// TIA Portal project "Banda_Asamblare" (V15.1)

(* hardware
DEVICE "S71500/ET200MP station_1"  S7-1500 station
   slot 0: "Rail_0"  Rack  6ES7 590-1***0-0AA0
   slot 1: "PLC_1"  CPU 1513-1 PN  6ES7 513-1AL02-0AB0  V2.6
      slot 3: "CPU display_1"  6ES7591-1AA00-0AA0
DEVICE "HMI_1"  KTP900 Basic PN
   slot 0: "HMI_1"  KTP900 Basic PN  6AV2 123-2JB03-0AX0  15.1.0.0
   slot 1: "HMI_RT_1"  KTP900 Basic PN  6AV2 123-2JB03-0AX0  15.1.0.0
   slot 5: "HMI_1.IE_CP_1"  PROFINET Interface  15.0.1.0
      slot 1: "PROFINET Interface_1"  PROFINET Interface
         slot 1: "Port_1"  Port
*)

// ===== PLC "PLC_1"  CPU 1513-1 PN =====

VAR_GLOBAL   // PLC tag table "Default tag table"
   "Clock_Byte" AT %MB0 : Byte;
   "Clock_10Hz" AT %M0.0 : Bool;
   "Clock_5Hz" AT %M0.1 : Bool;
   "Clock_2.5Hz" AT %M0.2 : Bool;
   "Clock_2Hz" AT %M0.3 : Bool;
   "Clock_1.25Hz" AT %M0.4 : Bool;
   "Clock_1Hz" AT %M0.5 : Bool;
   "Clock_0.625Hz" AT %M0.6 : Bool;
   "Clock_0.5Hz" AT %M0.7 : Bool;
END_VAR

DATA_BLOCK "Alarme"   // DB1
{ S7_Optimized_Access := 'TRUE' }
VERSION : 0.1
   VAR
      alarme_vect : Array[0..15] of Bool;
      alarme_gather : Word;
   END_VAR
BEGIN
END_DATA_BLOCK

DATA_BLOCK "Avarii"   // DB2
{ S7_Optimized_Access := 'TRUE' }
VERSION : 0.1
   VAR
      avarie_start : Bool;
      avarie_cuptor : Bool;
      avarie_aplatizor : Bool;
      avarie_forme : Bool;
      avarie_taiere : Bool;
      avarie_curatare : Bool;
      avarie_general : Bool;
      container1_plin : Bool;
      container2_plin : Bool;
      container3_plin : Bool;
      container_plin_general : Bool;
      limite_containere : Bool;
   END_VAR
BEGIN
END_DATA_BLOCK

DATA_BLOCK "Mecanisme"   // DB3
{ S7_Optimized_Access := 'TRUE' }
VERSION : 0.1
   VAR
      block_start : Bool;
      punere_block_material : Bool;
      cuptor : Bool;
      temperatura_cuptor : Real;
      "temperatura dorita la cuptor" : Real;
      temp_dorita_atinsa : Bool;
      aplatizor : Bool;
      forma : UInt;
      ajuns_la_forma1 : Bool;
      ajuns_la_forma2 : Bool;
      ajuns_la_forma3 : Bool;
      taiere1 : Bool;
      taiere2 : Bool;
      taiere3 : Bool;
      curatare1 : Bool;
      curatare2 : Bool;
      curatare3 : Bool;
      container_f1 : UInt;
      container_f2 : UInt;
      container_f3 : UInt;
      servo : UInt;
      limita_c1 : UInt;
      limita_c2 : UInt;
      limita_c3 : UInt;
      cond_cuptor : Bool;
   END_VAR
BEGIN
END_DATA_BLOCK

DATA_BLOCK "Butoane"   // DB4
{ S7_Optimized_Access := 'TRUE' }
VERSION : 0.1
   VAR
      btn_start : Bool;
      btn_esd : Bool;
      btn_stop : Bool;
      reset_esd : Bool;
      pornire : Bool;
      esd : Bool;
      "blocare_start_pe timer" : Bool;
      mentinere_timer_punere_material : Bool;
      "reset avarii" : Bool;
      timer_oprit : Bool;
      golire_c1 : Bool;
      golire_c2 : Bool;
      golire_c3 : Bool;
   END_VAR
BEGIN
END_DATA_BLOCK

DATA_BLOCK "Benzi"   // DB5
{ S7_Optimized_Access := 'TRUE' }
VERSION : 0.1
   VAR
      plecat_b1 : Bool;
      plecat_b2 : Bool;
      plecat_b3 : Bool;
      plecat_b41 : Bool;
      plecat_b42 : Bool;
      plecat_b43 : Bool;
      plecat_b51 : Bool;
      plecat_b52 : Bool;
      plecat_b53 : Bool;
      plecat_b61 : Bool;
      plecat_b62 : Bool;
      plecat_b63 : Bool;
   END_VAR
BEGIN
END_DATA_BLOCK

DATA_BLOCK "Comenzi_DB"   // DB7
{ S7_Optimized_Access := 'TRUE' }
VERSION : 0.1
// stored: InstanceOfName Comenzi
"Comenzi"
BEGIN
END_DATA_BLOCK

DATA_BLOCK "Banda_DB"   // DB8
{ S7_Optimized_Access := 'TRUE' }
VERSION : 0.1
// stored: InstanceOfName Banda
"Banda"
BEGIN
END_DATA_BLOCK

DATA_BLOCK "rising edges"   // DB9
{ S7_Optimized_Access := 'TRUE' }
VERSION : 0.1
   VAR
      re1 : Bool;
      re2 : Bool;
      re3 : Bool;
      re4 : Bool;
      re5 : Bool;
      re6 : Bool;
      re7 : Bool;
      re8 : Bool;
   END_VAR
BEGIN
END_DATA_BLOCK

DATA_BLOCK "Simulare_DB"   // DB13
{ S7_Optimized_Access := 'TRUE' }
VERSION : 0.1
// stored: InstanceOfName Simulare
"Simulare"
BEGIN
END_DATA_BLOCK

FUNCTION_BLOCK "Simulare"   // FB1, LAD
{ S7_Optimized_Access := 'TRUE' }
VERSION : 0.1
   VAR_INPUT
      btn_pornire : Bool;
      b1_plecat : Bool;
      b2_plecat : Bool;
      b3_plecat : Bool;
      b41_plecat : Bool;
      b42_plecat : Bool;
      b43_plecat : Bool;
      b51_plecat : Bool;
      b52_plecat : Bool;
      b53_plecat : Bool;
      b61_plecat : Bool;
      b62_plecat : Bool;
      b63_plecat : Bool;
      cond_cuptor : Bool;
      forma : UInt;
   END_VAR
   VAR_OUTPUT
      cuptor_pornit : Bool;
      aplatizor_pornit : Bool;
      forma1 : Bool;
      forma2 : Bool;
      forma3 : Bool;
      taiere1 : Bool;
      taiere2 : Bool;
      taiere3 : Bool;
      curatare1 : Bool;
      curatare2 : Bool;
      curatare3 : Bool;
      container1 : UInt;
      container2 : UInt;
      container3 : UInt;
      servo : UInt;
   END_VAR
   VAR_IN_OUT
      pune_material : Bool;
      btn_golire1 : Bool;
      btn_golire2 : Bool;
      btn_golire3 : Bool;
      temp_cuptor : Real;
   END_VAR
   VAR
      re1 : Bool;
      re2 : Bool;
      re3 : Bool;
      re4 : Bool;
      re5 : Bool;
      "timer reset punere material" : TON_TIME;
      mentinere_timer_material : Bool;
      timer_aplatizare : TON_TIME;
      "tiimer forma" : TON_TIME;
      "timer taiere1" : TON_TIME;
      "timer taiere2" : TON_TIME;
      "timer taiere3" : TON_TIME;
      "timer curatare1" : TON_TIME;
      "timer curatare 2" : TON_TIME;
      "timer curatare 3" : TON_TIME;
      "reset golire1" : TON_TIME;
      "reset golire 2" : TON_TIME;
      "reset golire 3" : TON_TIME;
   END_VAR
   VAR_TEMP   // added for the SCL form of the ladder/FBD networks
      _w1 : Bool;
      _w2 : Bool;
      _w3 : Bool;
   END_VAR
BEGIN

REGION Network 1: pune un block de material pe banda
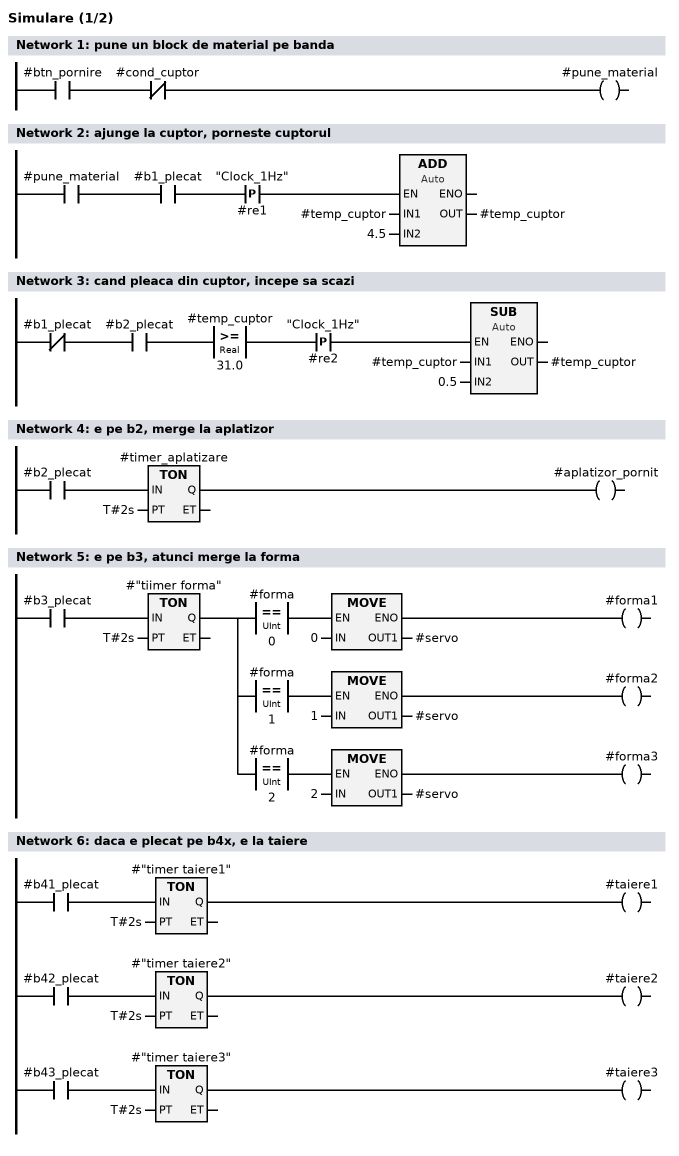
   RUNG wire#powerrail
      Contact( #btn_pornire )
      I_Contact( #cond_cuptor )
      Coil( #pune_material )
   END_RUNG
   // the same network as SCL:
   #pune_material := #btn_pornire AND NOT #cond_cuptor;
END_REGION

REGION Network 2: ajunge la cuptor, porneste cuptorul
   RUNG wire#powerrail
      Contact( #pune_material )
      Contact( #b1_plecat )
      P_Contact(operand := "Clock_1Hz", bit := #re1)
      Add(in1 := #temp_cuptor, in2 := 4.5, out => #temp_cuptor)
   END_RUNG
   // the same network as SCL:
   #_w1 := #pune_material AND #b1_plecat AND "Clock_1Hz" AND NOT #re1;   // rising edge of "Clock_1Hz"
   #re1 := "Clock_1Hz";
   IF #_w1 THEN #temp_cuptor := #temp_cuptor + 4.5; END_IF;
END_REGION

REGION Network 3: cand pleaca din cuptor, incepe sa scazi
   RUNG wire#powerrail
      I_Contact( #b1_plecat )
      Contact( #b2_plecat )
      { S7_Templates := "SrcType := Real" } GE_Contact(in1 := #temp_cuptor, in2 := 31.0)
      P_Contact(operand := "Clock_1Hz", bit := #re2)
      Sub(in1 := #temp_cuptor, in2 := 0.5, out => #temp_cuptor)
   END_RUNG
   // the same network as SCL:
   #_w1 := NOT #b1_plecat AND #b2_plecat AND (#temp_cuptor >= 31.0) AND "Clock_1Hz" AND NOT #re2;   // rising edge of "Clock_1Hz"
   #re2 := "Clock_1Hz";
   IF #_w1 THEN #temp_cuptor := #temp_cuptor - 0.5; END_IF;
END_REGION

REGION Network 4: e pe b2, merge la aplatizor
   #timer_aplatizare(IN := #b2_plecat, PT := T#2s);   // TON
   #aplatizor_pornit := #timer_aplatizare.Q;
END_REGION

REGION Network 5: e pe b3, atunci merge la forma
   #"tiimer forma"(IN := #b3_plecat, PT := T#2s);   // TON
   #_w1 := #"tiimer forma".Q AND (#forma = 0);
   IF #_w1 THEN #servo := 0; END_IF;
   #forma1 := #_w1;
   #_w2 := #"tiimer forma".Q AND (#forma = 1);
   IF #_w2 THEN #servo := 1; END_IF;
   #forma2 := #_w2;
   #_w3 := #"tiimer forma".Q AND (#forma = 2);
   IF #_w3 THEN #servo := 2; END_IF;
   #forma3 := #_w3;
END_REGION

REGION Network 6: daca e plecat pe b4x, e la taiere
   #"timer taiere1"(IN := #b41_plecat, PT := T#2s);   // TON
   #taiere1 := #"timer taiere1".Q;
   #"timer taiere2"(IN := #b42_plecat, PT := T#2s);   // TON
   #taiere2 := #"timer taiere2".Q;
   #"timer taiere3"(IN := #b43_plecat, PT := T#2s);   // TON
   #taiere3 := #"timer taiere3".Q;
END_REGION

REGION Network 7: daca e pe banda b5x, sa dea drumul la curatari
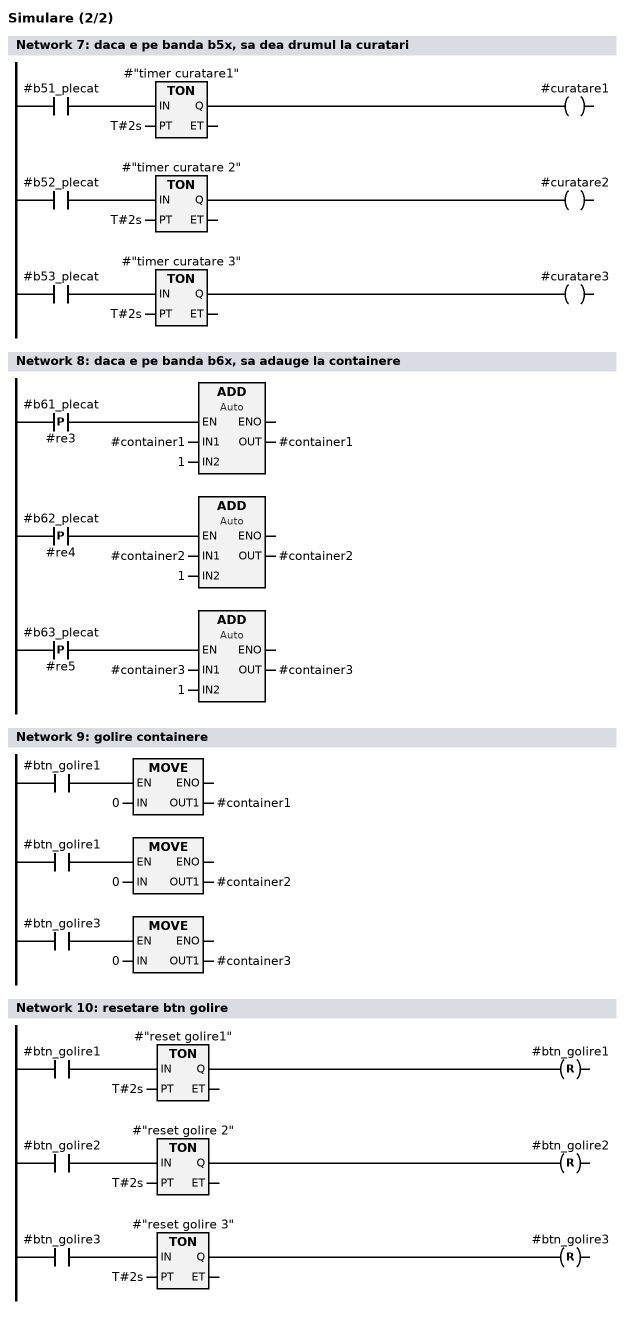
   #"timer curatare1"(IN := #b51_plecat, PT := T#2s);   // TON
   #curatare1 := #"timer curatare1".Q;
   #"timer curatare 2"(IN := #b52_plecat, PT := T#2s);   // TON
   #curatare2 := #"timer curatare 2".Q;
   #"timer curatare 3"(IN := #b53_plecat, PT := T#2s);   // TON
   #curatare3 := #"timer curatare 3".Q;
END_REGION

REGION Network 8: daca e pe banda b6x, sa adauge la containere
   RUNG wire#powerrail
      P_Contact(operand := #b61_plecat, bit := #re3)
      Add(in1 := #container1, in2 := 1, out => #container1)
   END_RUNG
   RUNG wire#powerrail
      P_Contact(operand := #b62_plecat, bit := #re4)
      Add(in1 := #container2, in2 := 1, out => #container2)
   END_RUNG
   RUNG wire#powerrail
      P_Contact(operand := #b63_plecat, bit := #re5)
      Add(in1 := #container3, in2 := 1, out => #container3)
   END_RUNG
   // the same network as SCL:
   #_w1 := #b61_plecat AND NOT #re3;   // rising edge of #b61_plecat
   #re3 := #b61_plecat;
   IF #_w1 THEN #container1 := #container1 + 1; END_IF;
   #_w2 := #b62_plecat AND NOT #re4;   // rising edge of #b62_plecat
   #re4 := #b62_plecat;
   IF #_w2 THEN #container2 := #container2 + 1; END_IF;
   #_w3 := #b63_plecat AND NOT #re5;   // rising edge of #b63_plecat
   #re5 := #b63_plecat;
   IF #_w3 THEN #container3 := #container3 + 1; END_IF;
END_REGION

REGION Network 9: golire containere
   RUNG wire#powerrail
      Contact( #btn_golire1 )
      Move(in := 0, out1 => #container1)
   END_RUNG
   RUNG wire#powerrail
      Contact( #btn_golire1 )
      Move(in := 0, out1 => #container2)
   END_RUNG
   RUNG wire#powerrail
      Contact( #btn_golire3 )
      Move(in := 0, out1 => #container3)
   END_RUNG
   // the same network as SCL:
   IF #btn_golire1 THEN
       #container1 := 0;
       #container2 := 0;
   END_IF;
   IF #btn_golire3 THEN #container3 := 0; END_IF;
END_REGION

REGION Network 10: resetare btn golire
   #"reset golire1"(IN := #btn_golire1, PT := T#2s);   // TON
   IF #"reset golire1".Q THEN #btn_golire1 := FALSE; END_IF;
   #"reset golire 2"(IN := #btn_golire2, PT := T#2s);   // TON
   IF #"reset golire 2".Q THEN #btn_golire2 := FALSE; END_IF;
   #"reset golire 3"(IN := #btn_golire3, PT := T#2s);   // TON
   IF #"reset golire 3".Q THEN #btn_golire3 := FALSE; END_IF;
END_REGION
END_FUNCTION_BLOCK

FUNCTION_BLOCK "Comenzi"   // FB2, LAD
{ S7_Optimized_Access := 'TRUE' }
VERSION : 0.1
   VAR_INPUT
      temp_cuptor : Real;
      temp_dorita : Real;
      pune_material : Bool;
      aplatizor_pornit : Bool;
      forma1 : Bool;
      forma2 : Bool;
      forma3 : Bool;
      taiere1 : Bool;
      taiere2 : Bool;
      taiere3 : Bool;
      curatare1 : Bool;
      curatare2 : Bool;
      curatare3 : Bool;
   END_VAR
   VAR_OUTPUT
      b1_plecat : Bool;
      b2_plecat : Bool;
      b3_plecat : Bool;
      b41_plecat : Bool;
      b42_plecat : Bool;
      b43_plecat : Bool;
      b51_plecat : Bool;
      b52_plecat : Bool;
      b53_plecat : Bool;
      b61_plecat : Bool;
      b62_plecat : Bool;
      b63_plecat : Bool;
      cond_cuptor : Bool;
   END_VAR
   VAR
      "timer plecare b1" : TON_TIME;
      incc : Int;
      edg : Bool;
   END_VAR
BEGIN

REGION Network 1: pleaca spre cuptor
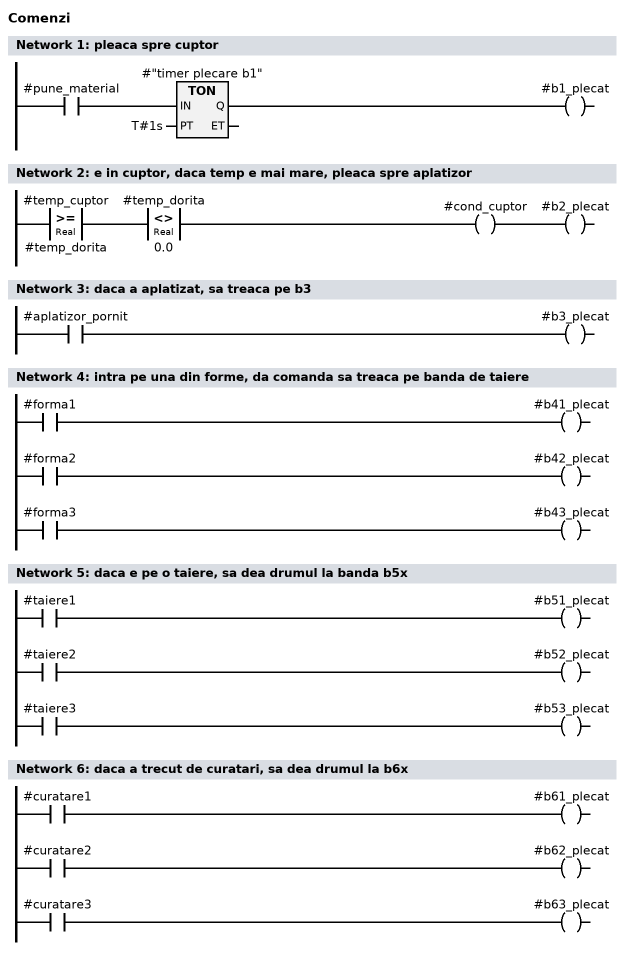
   #"timer plecare b1"(IN := #pune_material, PT := T#1s);   // TON
   #b1_plecat := #"timer plecare b1".Q;
END_REGION

REGION Network 2: e in cuptor, daca temp e mai mare, pleaca spre aplatizor
   RUNG wire#powerrail
      { S7_Templates := "SrcType := Real" } GE_Contact(in1 := #temp_cuptor, in2 := #temp_dorita)
      { S7_Templates := "SrcType := Real" } NE_Contact(in1 := #temp_dorita, in2 := 0.0)
      Coil( #cond_cuptor )
      Coil( #b2_plecat )
   END_RUNG
   // the same network as SCL:
   #cond_cuptor := (#temp_cuptor >= #temp_dorita) AND (#temp_dorita <> 0.0);
   #b2_plecat := #cond_cuptor;
END_REGION

REGION Network 3: daca a aplatizat, sa treaca pe b3
   RUNG wire#powerrail
      Contact( #aplatizor_pornit )
      Coil( #b3_plecat )
   END_RUNG
   // the same network as SCL:
   #b3_plecat := #aplatizor_pornit;
END_REGION

REGION Network 4: intra pe una din forme, da comanda sa treaca pe banda de taiere
   RUNG wire#powerrail
      Contact( #forma1 )
      Coil( #b41_plecat )
   END_RUNG
   RUNG wire#powerrail
      Contact( #forma2 )
      Coil( #b42_plecat )
   END_RUNG
   RUNG wire#powerrail
      Contact( #forma3 )
      Coil( #b43_plecat )
   END_RUNG
   // the same network as SCL:
   #b41_plecat := #forma1;
   #b42_plecat := #forma2;
   #b43_plecat := #forma3;
END_REGION

REGION Network 5: daca e pe o taiere, sa dea drumul la banda b5x
   RUNG wire#powerrail
      Contact( #taiere1 )
      Coil( #b51_plecat )
   END_RUNG
   RUNG wire#powerrail
      Contact( #taiere2 )
      Coil( #b52_plecat )
   END_RUNG
   RUNG wire#powerrail
      Contact( #taiere3 )
      Coil( #b53_plecat )
   END_RUNG
   // the same network as SCL:
   #b51_plecat := #taiere1;
   #b52_plecat := #taiere2;
   #b53_plecat := #taiere3;
END_REGION

REGION Network 6: daca a trecut de curatari, sa dea drumul la b6x
   RUNG wire#powerrail
      Contact( #curatare1 )
      Coil( #b61_plecat )
   END_RUNG
   RUNG wire#powerrail
      Contact( #curatare2 )
      Coil( #b62_plecat )
   END_RUNG
   RUNG wire#powerrail
      Contact( #curatare3 )
      Coil( #b63_plecat )
   END_RUNG
   // the same network as SCL:
   #b61_plecat := #curatare1;
   #b62_plecat := #curatare2;
   #b63_plecat := #curatare3;
END_REGION
END_FUNCTION_BLOCK

FUNCTION_BLOCK "Banda"   // FB3, LAD
{ S7_Optimized_Access := 'TRUE' }
VERSION : 0.1
   VAR_INPUT
      temperatura_dorita : Real := 0.0;
      forma : UInt := 0;
      stop : Bool;
      start : Bool;
      limita_container1 : UInt;
      limita_container2 : UInt;
      limita_container3 : UInt;
   END_VAR
   VAR_OUTPUT
      cuptor : Bool;
      aplatizor : Bool;
      taiere1 : Bool;
      taiere2 : Bool;
      taiere3 : Bool;
      curatare1 : Bool;
      curatare2 : Bool;
      curatare3 : Bool;
   END_VAR
   VAR_IN_OUT
      golire_c1 : Bool;
      golire_c2 : Bool;
      golire_c3 : Bool;
      container1 : UInt;
      container2 : UInt;
      container3 : UInt;
      temperatura_cuptor : Real;
      reset_esd : Bool;
      btn_esd : Bool;
      btn_reset_avarii : Bool;
      avarie_start : Bool;
      avarie_cuptor : Bool;
      avarie_aplatizor : Bool;
      avarie_forma : Bool;
      avarie_taiere : Bool;
      avarie_curatare : Bool;
   END_VAR
   VAR
      esd : Bool;
      limite_containere : Bool;
      Avarii_generale : Bool;
      container_plin : Bool;
      pornire : Bool;
      alarme_gather : Word;
      alarme_vect : Array[0..15] of Bool;
      punere_block : Bool;
      ajuns_forma1 : Bool;
      ajuns_forma2 : Bool;
      ajuns_forma3 : Bool;
      plecat_b1 : Bool;
      plecat_b2 : Bool;
      plecat_b3 : Bool;
      plecat_b41 : Bool;
      plecat_b42 : Bool;
      plecat_b43 : Bool;
      plecar_b51 : Bool;
      plecar_b52 : Bool;
      plecar_b53 : Bool;
      plecat_b61 : Bool;
      plecat_b62 : Bool;
      plecat_b63 : Bool;
      cond_cuptor : Bool;
      servo : UInt;
      reset_esd_timer : TON_TIME;
      plin_container1 : Bool;
      plin_container2 : Bool;
      plin_container3 : Bool;
   END_VAR
BEGIN

REGION Network 1: buton start
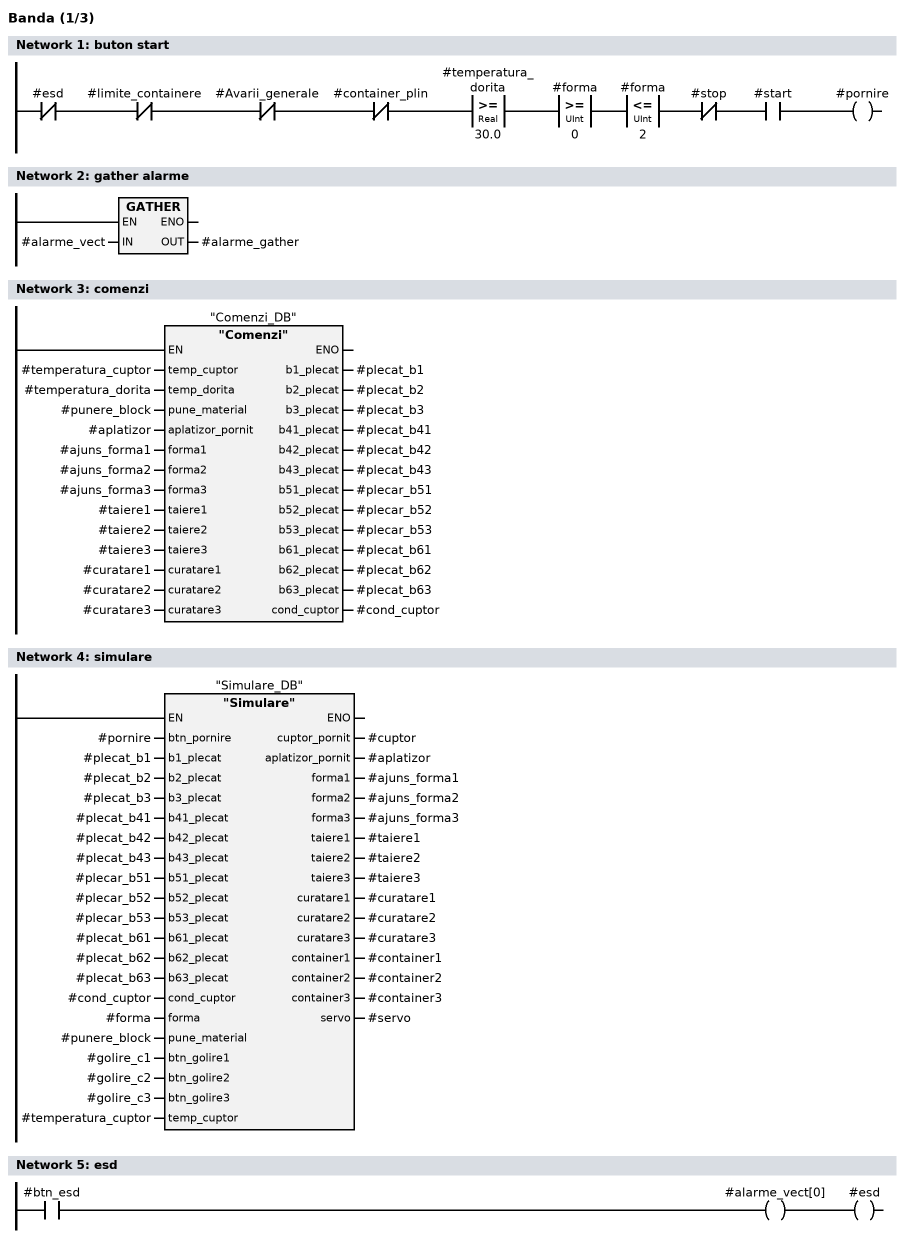
   RUNG wire#powerrail
      I_Contact( #esd )
      I_Contact( #limite_containere )
      I_Contact( #Avarii_generale )
      I_Contact( #container_plin )
      { S7_Templates := "SrcType := Real" } GE_Contact(in1 := #temperatura_dorita, in2 := 30.0)
      { S7_Templates := "SrcType := UInt" } GE_Contact(in1 := #forma, in2 := 0)
      { S7_Templates := "SrcType := UInt" } LE_Contact(in1 := #forma, in2 := 2)
      I_Contact( #stop )
      Contact( #start )
      Coil( #pornire )
   END_RUNG
   // the same network as SCL:
   #pornire := NOT #esd AND NOT #limite_containere AND NOT #Avarii_generale AND NOT #container_plin AND (#temperatura_dorita >= 30.0) AND (#forma >= 0) AND (#forma <= 2) AND NOT #stop AND #start;
END_REGION

REGION Network 2: gather alarme
   GATHER(IN := #alarme_vect, OUT => #alarme_gather);
END_REGION

REGION Network 3: comenzi
   RUNG wire#powerrail
      "Comenzi_DB"(temp_cuptor := #temperatura_cuptor, temp_dorita := #temperatura_dorita, pune_material := #punere_block, aplatizor_pornit := #aplatizor, forma1 := #ajuns_forma1, forma2 := #ajuns_forma2, forma3 := #ajuns_forma3, taiere1 := #taiere1, taiere2 := #taiere2, taiere3 := #taiere3, curatare1 := #curatare1, curatare2 := #curatare2, curatare3 := #curatare3, b1_plecat => #plecat_b1, b2_plecat => #plecat_b2, b3_plecat => #plecat_b3, b41_plecat => #plecat_b41, b42_plecat => #plecat_b42, b43_plecat => #plecat_b43, b51_plecat => #plecar_b51, b52_plecat => #plecar_b52, b53_plecat => #plecar_b53, b61_plecat => #plecat_b61, b62_plecat => #plecat_b62, b63_plecat => #plecat_b63, cond_cuptor => #cond_cuptor)
   END_RUNG
   // the same network as SCL:
   "Comenzi_DB"(temp_cuptor := #temperatura_cuptor,   // "Comenzi"
                temp_dorita := #temperatura_dorita,
                pune_material := #punere_block,
                aplatizor_pornit := #aplatizor,
                forma1 := #ajuns_forma1,
                forma2 := #ajuns_forma2,
                forma3 := #ajuns_forma3,
                taiere1 := #taiere1,
                taiere2 := #taiere2,
                taiere3 := #taiere3,
                curatare1 := #curatare1,
                curatare2 := #curatare2,
                curatare3 := #curatare3,
                b1_plecat => #plecat_b1,
                b2_plecat => #plecat_b2,
                b3_plecat => #plecat_b3,
                b41_plecat => #plecat_b41,
                b42_plecat => #plecat_b42,
                b43_plecat => #plecat_b43,
                b51_plecat => #plecar_b51,
                b52_plecat => #plecar_b52,
                b53_plecat => #plecar_b53,
                b61_plecat => #plecat_b61,
                b62_plecat => #plecat_b62,
                b63_plecat => #plecat_b63,
                cond_cuptor => #cond_cuptor);
END_REGION

REGION Network 4: simulare
   RUNG wire#powerrail
      "Simulare_DB"(btn_pornire := #pornire, b1_plecat := #plecat_b1, b2_plecat := #plecat_b2, b3_plecat := #plecat_b3, b41_plecat := #plecat_b41, b42_plecat := #plecat_b42, b43_plecat := #plecat_b43, b51_plecat := #plecar_b51, b52_plecat := #plecar_b52, b53_plecat := #plecar_b53, b61_plecat := #plecat_b61, b62_plecat := #plecat_b62, b63_plecat := #plecat_b63, cond_cuptor := #cond_cuptor, forma := #forma, pune_material := #punere_block, btn_golire1 := #golire_c1, btn_golire2 := #golire_c2, btn_golire3 := #golire_c3, temp_cuptor := #temperatura_cuptor, cuptor_pornit => #cuptor, aplatizor_pornit => #aplatizor, forma1 => #ajuns_forma1, forma2 => #ajuns_forma2, forma3 => #ajuns_forma3, taiere1 => #taiere1, taiere2 => #taiere2, taiere3 => #taiere3, curatare1 => #curatare1, curatare2 => #curatare2, curatare3 => #curatare3, container1 => #container1, container2 => #container2, container3 => #container3, servo => #servo)
   END_RUNG
   // the same network as SCL:
   "Simulare_DB"(btn_pornire := #pornire,   // "Simulare"
                 b1_plecat := #plecat_b1,
                 b2_plecat := #plecat_b2,
                 b3_plecat := #plecat_b3,
                 b41_plecat := #plecat_b41,
                 b42_plecat := #plecat_b42,
                 b43_plecat := #plecat_b43,
                 b51_plecat := #plecar_b51,
                 b52_plecat := #plecar_b52,
                 b53_plecat := #plecar_b53,
                 b61_plecat := #plecat_b61,
                 b62_plecat := #plecat_b62,
                 b63_plecat := #plecat_b63,
                 cond_cuptor := #cond_cuptor,
                 forma := #forma,
                 pune_material := #punere_block,
                 btn_golire1 := #golire_c1,
                 btn_golire2 := #golire_c2,
                 btn_golire3 := #golire_c3,
                 temp_cuptor := #temperatura_cuptor,
                 cuptor_pornit => #cuptor,
                 aplatizor_pornit => #aplatizor,
                 forma1 => #ajuns_forma1,
                 forma2 => #ajuns_forma2,
                 forma3 => #ajuns_forma3,
                 taiere1 => #taiere1,
                 taiere2 => #taiere2,
                 taiere3 => #taiere3,
                 curatare1 => #curatare1,
                 curatare2 => #curatare2,
                 curatare3 => #curatare3,
                 container1 => #container1,
                 container2 => #container2,
                 container3 => #container3,
                 servo => #servo);
END_REGION

REGION Network 5: esd
   RUNG wire#powerrail
      Contact( #btn_esd )
      Coil( #alarme_vect[0] )
      Coil( #esd )
   END_RUNG
   // the same network as SCL:
   #alarme_vect[0] := #btn_esd;
   #esd := #btn_esd;
END_REGION

REGION Network 6: reset esd
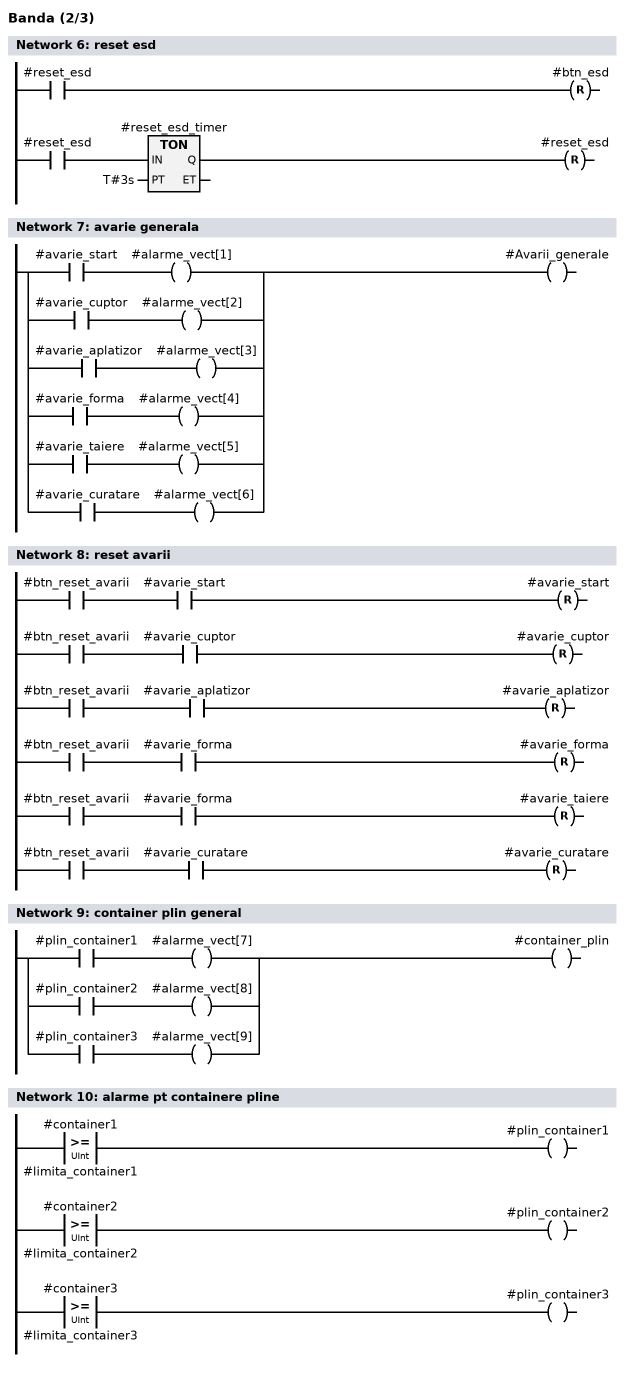
   IF #reset_esd THEN #btn_esd := FALSE; END_IF;
   #reset_esd_timer(IN := #reset_esd, PT := T#3s);   // TON
   IF #reset_esd_timer.Q THEN #reset_esd := FALSE; END_IF;
END_REGION

REGION Network 7: avarie generala
   RUNG wire#powerrail
      Contact( #avarie_start )
      Coil( #alarme_vect[1] )
      wire#w1
      Coil( #Avarii_generale )
   END_RUNG
   RUNG wire#powerrail
      Contact( #avarie_cuptor )
      Coil( #alarme_vect[2] )
   END_RUNG wire#w1
   RUNG wire#powerrail
      Contact( #avarie_aplatizor )
      Coil( #alarme_vect[3] )
   END_RUNG wire#w1
   RUNG wire#powerrail
      Contact( #avarie_forma )
      Coil( #alarme_vect[4] )
   END_RUNG wire#w1
   RUNG wire#powerrail
      Contact( #avarie_taiere )
      Coil( #alarme_vect[5] )
   END_RUNG wire#w1
   RUNG wire#powerrail
      Contact( #avarie_curatare )
      Coil( #alarme_vect[6] )
   END_RUNG wire#w1
   // the same network as SCL:
   #alarme_vect[1] := #avarie_start;
   #alarme_vect[2] := #avarie_cuptor;
   #alarme_vect[3] := #avarie_aplatizor;
   #alarme_vect[4] := #avarie_forma;
   #alarme_vect[5] := #avarie_taiere;
   #alarme_vect[6] := #avarie_curatare;
   #Avarii_generale := #avarie_start OR #avarie_cuptor OR #avarie_aplatizor OR #avarie_forma OR #avarie_taiere OR #avarie_curatare;
END_REGION

REGION Network 8: reset avarii
   RUNG wire#powerrail
      Contact( #btn_reset_avarii )
      Contact( #avarie_start )
      R_Coil( #avarie_start )
   END_RUNG
   RUNG wire#powerrail
      Contact( #btn_reset_avarii )
      Contact( #avarie_cuptor )
      R_Coil( #avarie_cuptor )
   END_RUNG
   RUNG wire#powerrail
      Contact( #btn_reset_avarii )
      Contact( #avarie_aplatizor )
      R_Coil( #avarie_aplatizor )
   END_RUNG
   RUNG wire#powerrail
      Contact( #btn_reset_avarii )
      Contact( #avarie_forma )
      R_Coil( #avarie_forma )
   END_RUNG
   RUNG wire#powerrail
      Contact( #btn_reset_avarii )
      Contact( #avarie_forma )
      R_Coil( #avarie_taiere )
   END_RUNG
   RUNG wire#powerrail
      Contact( #btn_reset_avarii )
      Contact( #avarie_curatare )
      R_Coil( #avarie_curatare )
   END_RUNG
   // the same network as SCL:
   IF #btn_reset_avarii AND #avarie_start THEN #avarie_start := FALSE; END_IF;
   IF #btn_reset_avarii AND #avarie_cuptor THEN #avarie_cuptor := FALSE; END_IF;
   IF #btn_reset_avarii AND #avarie_aplatizor THEN #avarie_aplatizor := FALSE; END_IF;
   IF #btn_reset_avarii AND #avarie_forma THEN #avarie_forma := FALSE; END_IF;
   IF #btn_reset_avarii AND #avarie_forma THEN #avarie_taiere := FALSE; END_IF;
   IF #btn_reset_avarii AND #avarie_curatare THEN #avarie_curatare := FALSE; END_IF;
END_REGION

REGION Network 9: container plin general
   RUNG wire#powerrail
      Contact( #plin_container1 )
      Coil( #alarme_vect[7] )
      wire#w1
      Coil( #container_plin )
   END_RUNG
   RUNG wire#powerrail
      Contact( #plin_container2 )
      Coil( #alarme_vect[8] )
   END_RUNG wire#w1
   RUNG wire#powerrail
      Contact( #plin_container3 )
      Coil( #alarme_vect[9] )
   END_RUNG wire#w1
   // the same network as SCL:
   #alarme_vect[7] := #plin_container1;
   #alarme_vect[8] := #plin_container2;
   #alarme_vect[9] := #plin_container3;
   #container_plin := #plin_container1 OR #plin_container2 OR #plin_container3;
END_REGION

REGION Network 10: alarme pt containere pline
   RUNG wire#powerrail
      { S7_Templates := "SrcType := UInt" } GE_Contact(in1 := #container1, in2 := #limita_container1)
      Coil( #plin_container1 )
   END_RUNG
   RUNG wire#powerrail
      { S7_Templates := "SrcType := UInt" } GE_Contact(in1 := #container2, in2 := #limita_container2)
      Coil( #plin_container2 )
   END_RUNG
   RUNG wire#powerrail
      { S7_Templates := "SrcType := UInt" } GE_Contact(in1 := #container3, in2 := #limita_container3)
      Coil( #plin_container3 )
   END_RUNG
   // the same network as SCL:
   #plin_container1 := #container1 >= #limita_container1;
   #plin_container2 := #container2 >= #limita_container2;
   #plin_container3 := #container3 >= #limita_container3;
END_REGION

REGION Network 11: limite containere
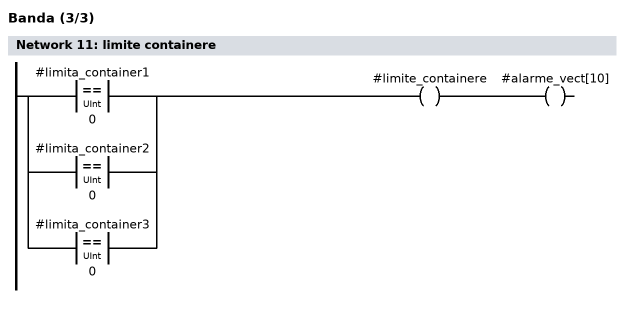
   RUNG wire#powerrail
      { S7_Templates := "SrcType := UInt" } EQ_Contact(in1 := #limita_container1, in2 := 0)
      wire#w1
      Coil( #limite_containere )
      Coil( #alarme_vect[10] )
   END_RUNG
   RUNG wire#powerrail
      { S7_Templates := "SrcType := UInt" } EQ_Contact(in1 := #limita_container2, in2 := 0)
   END_RUNG wire#w1
   RUNG wire#powerrail
      { S7_Templates := "SrcType := UInt" } EQ_Contact(in1 := #limita_container3, in2 := 0)
   END_RUNG wire#w1
   // the same network as SCL:
   #limite_containere := (#limita_container1 = 0) OR (#limita_container2 = 0) OR (#limita_container3 = 0);
   #alarme_vect[10] := #limite_containere;
END_REGION
END_FUNCTION_BLOCK

ORGANIZATION_BLOCK "Main"   // OB1, LAD, ProgramCycle
TITLE = "Main Program Sweep (Cycle)"
{ S7_Optimized_Access := 'TRUE' }
VERSION : 0.1
   VAR_INPUT
      Initial_Call : Bool;   // Initial call of this OB
      Remanence : Bool;   // =True, if remanent data are available
   END_VAR
BEGIN

REGION Network 1
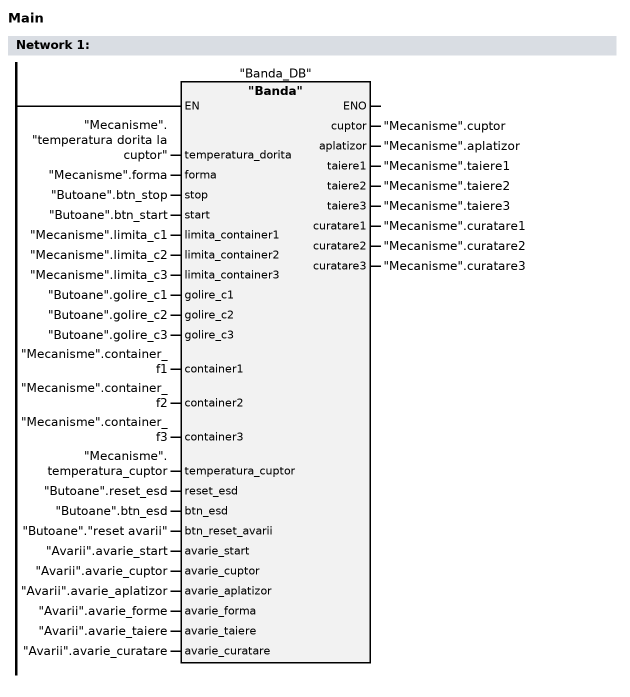
   RUNG wire#powerrail
      "Banda_DB"(temperatura_dorita := "Mecanisme"."temperatura dorita la cuptor", forma := "Mecanisme".forma, stop := "Butoane".btn_stop, start := "Butoane".btn_start, limita_container1 := "Mecanisme".limita_c1, limita_container2 := "Mecanisme".limita_c2, limita_container3 := "Mecanisme".limita_c3, golire_c1 := "Butoane".golire_c1, golire_c2 := "Butoane".golire_c2, golire_c3 := "Butoane".golire_c3, container1 := "Mecanisme".container_f1, container2 := "Mecanisme".container_f2, container3 := "Mecanisme".container_f3, temperatura_cuptor := "Mecanisme".temperatura_cuptor, reset_esd := "Butoane".reset_esd, btn_esd := "Butoane".btn_esd, btn_reset_avarii := "Butoane"."reset avarii", avarie_start := "Avarii".avarie_start, avarie_cuptor := "Avarii".avarie_cuptor, avarie_aplatizor := "Avarii".avarie_aplatizor, avarie_forma := "Avarii".avarie_forme, avarie_taiere := "Avarii".avarie_taiere, avarie_curatare := "Avarii".avarie_curatare, cuptor => "Mecanisme".cuptor, aplatizor => "Mecanisme".aplatizor, taiere1 => "Mecanisme".taiere1, taiere2 => "Mecanisme".taiere2, taiere3 => "Mecanisme".taiere3, curatare1 => "Mecanisme".curatare1, curatare2 => "Mecanisme".curatare2, curatare3 => "Mecanisme".curatare3)
   END_RUNG
   // the same network as SCL:
   "Banda_DB"(temperatura_dorita := "Mecanisme"."temperatura dorita la cuptor",   // "Banda"
              forma := "Mecanisme".forma,
              stop := "Butoane".btn_stop,
              start := "Butoane".btn_start,
              limita_container1 := "Mecanisme".limita_c1,
              limita_container2 := "Mecanisme".limita_c2,
              limita_container3 := "Mecanisme".limita_c3,
              golire_c1 := "Butoane".golire_c1,
              golire_c2 := "Butoane".golire_c2,
              golire_c3 := "Butoane".golire_c3,
              container1 := "Mecanisme".container_f1,
              container2 := "Mecanisme".container_f2,
              container3 := "Mecanisme".container_f3,
              temperatura_cuptor := "Mecanisme".temperatura_cuptor,
              reset_esd := "Butoane".reset_esd,
              btn_esd := "Butoane".btn_esd,
              btn_reset_avarii := "Butoane"."reset avarii",
              avarie_start := "Avarii".avarie_start,
              avarie_cuptor := "Avarii".avarie_cuptor,
              avarie_aplatizor := "Avarii".avarie_aplatizor,
              avarie_forma := "Avarii".avarie_forme,
              avarie_taiere := "Avarii".avarie_taiere,
              avarie_curatare := "Avarii".avarie_curatare,
              cuptor => "Mecanisme".cuptor,
              aplatizor => "Mecanisme".aplatizor,
              taiere1 => "Mecanisme".taiere1,
              taiere2 => "Mecanisme".taiere2,
              taiere3 => "Mecanisme".taiere3,
              curatare1 => "Mecanisme".curatare1,
              curatare2 => "Mecanisme".curatare2,
              curatare3 => "Mecanisme".curatare3);
END_REGION
END_ORGANIZATION_BLOCK

(* ===== HMI "HMI_RT_1" =====
system functions are stored by id; their names below are inferred from use
connection "HMI_Connection_1": ETHERNET, SMART_S7_1500_OMS

HMI tags "Default tag table"
   "Tag_ScreenNumber" : UInt, internal
   "Alarme_alarme_gather" : Word = PLC Alarme.alarme_gather, 1 s
   "Avarii_avarie_start" : Bool = PLC Avarii.avarie_start, 1 s
   "Avarii_avarie_cuptor" : Bool = PLC Avarii.avarie_cuptor, 1 s
   "Avarii_avarie_aplatizor" : Bool = PLC Avarii.avarie_aplatizor, 1 s
   "Avarii_avarie_forme" : Bool = PLC Avarii.avarie_forme, 1 s
   "Avarii_avarie_taiere" : Bool = PLC Avarii.avarie_taiere, 1 s
   "Avarii_avarie_curatare" : Bool = PLC Avarii.avarie_curatare, 1 s
   "Butoane_reset avarii" : Bool = PLC Butoane."reset avarii", 1 s
   "Mecanisme_forma" : UInt = PLC Mecanisme.forma, 1 s
   "Butoane_btn_start" : Bool = PLC Butoane.btn_start, 1 s
   "Butoane_esd" : Bool = PLC Butoane.esd, 1 s
   "Butoane_btn_esd" : Bool = PLC Butoane.btn_esd, 1 s
   "Butoane_reset_esd" : Bool = PLC Butoane.reset_esd, 1 s
   "Mecanisme_cuptor" : Bool = PLC Mecanisme.cuptor, 1 s
   "Butoane_golire_c1" : Bool = PLC Butoane.golire_c1, 1 s
   "Butoane_golire_c2" : Bool = PLC Butoane.golire_c2, 1 s
   "Butoane_golire_c3" : Bool = PLC Butoane.golire_c3, 1 s
   "Mecanisme_aplatizor" : Bool = PLC Mecanisme.aplatizor, 1 s
   "Mecanisme_taiere1" : Bool = PLC Mecanisme.taiere1, 1 s
   "Mecanisme_taiere2" : Bool = PLC Mecanisme.taiere2, 1 s
   "Mecanisme_taiere3" : Bool = PLC Mecanisme.taiere3, 1 s
   "Mecanisme_curatare1" : Bool = PLC Mecanisme.curatare1, 1 s
   "Mecanisme_curatare2" : Bool = PLC Mecanisme.curatare2, 1 s
   "Mecanisme_curatare3" : Bool = PLC Mecanisme.curatare3, 1 s
   "Mecanisme_container_f1" : UInt = PLC Mecanisme.container_f1, 1 s
   "Mecanisme_container_f2" : UInt = PLC Mecanisme.container_f2, 1 s
   "Mecanisme_container_f3" : UInt = PLC Mecanisme.container_f3, 1 s
   "Mecanisme_limita_c1" : UInt = PLC Mecanisme.limita_c1, 1 s
   "Mecanisme_limita_c2" : UInt = PLC Mecanisme.limita_c2, 1 s
   "Mecanisme_limita_c3" : UInt = PLC Mecanisme.limita_c3, 1 s
   "Comenzi_DB_temp_dorita" : Real = PLC Comenzi_DB.temp_dorita, 1 s
   "Comenzi_DB_temp_cuptor" : Real = PLC Comenzi_DB.temp_cuptor, 1 s
   "Mecanisme_temperatura dorita la cuptor" : Real = PLC Mecanisme."temperatura dorita la cuptor", 1 s
   "Mecanisme_temperatura_cuptor" : Real = PLC Mecanisme.temperatura_cuptor, 1 s
   "Butoane_btn_stop" : Bool = PLC Butoane.btn_stop, 1 s

discrete alarms
   1: 'Esd Apasat', class Errors, trigger "Alarme_alarme_gather" bit 0
   2: 'Avarie la Start', class Errors, trigger "Alarme_alarme_gather" bit 1
   3: 'Avarie la Cuptor', class Errors, trigger "Alarme_alarme_gather" bit 2
   4: 'Avarie la Aplatizor', class Errors, trigger "Alarme_alarme_gather" bit 3
   5: 'Avarie la Forme', class Errors, trigger "Alarme_alarme_gather" bit 4
   6: 'Avarie la Taiere', class Errors, trigger "Alarme_alarme_gather" bit 5
   7: 'Avarie la Curatare', class Errors, trigger "Alarme_alarme_gather" bit 6
   8: 'Container1 plin', class Errors, trigger "Alarme_alarme_gather" bit 7
   9: 'Container2 plin', class Errors, trigger "Alarme_alarme_gather" bit 8
   10: 'Container3 plin', class Errors, trigger "Alarme_alarme_gather" bit 9
   11: 'Limita la unul dintre containere nu este introdusa', class Errors, trigger "Alarme_alarme_gather" bit 10

text list "Forme": 0 'Forma1'; 1 'Forma2'; 2 'Forma3'

Template "Template_1" 800x480
   Button "Exit" at 722,440 size 55x39; TextOff 'Exit'; PictureOff "ExitRuntime_KTP900_Basic_PN_TR"; PictureOn "ExitRuntime_KTP900_Basic_PN_TR"
      on Release: StopRuntime(0)
   Button "Template_Button" at 622,440 size 55x39; TextOff 'Text'
   Button "Template_Button_1" at 522,440 size 55x39; TextOff 'Text'
   Button "Template_Button_2" at 422,440 size 55x39; TextOff 'Text'
   Button "Template_Button_3" at 322,440 size 55x39; TextOff 'Text'
   Button "Template_Button_4" at 222,440 size 55x39; TextOff 'Text'
   Button "Alarms" at 122,440 size 55x39; TextOff 'Alarms'; PictureOff "AlarmDisplay_KTP900_Basic_PN_TR"; PictureOn "AlarmDisplay_KTP900_Basic_PN_TR"
      on Release: function_ef3f5d25("Alarm window_1", -1)
   Button "Start screen" at 22,440 size 55x39; TextOff 'Start screen'; PictureOff "NavigateHome_KTP900_Basic_PN_TR"; PictureOn "NavigateHome_KTP900_Basic_PN_TR"
      on Release: ActivateScreen("Main", 0)
   SymbolicIOField "Symbolic_IO_Field_Screen" at 73,7 size 620x26; TextOff '0'; TextOn '1'; TextList "TextList_ScreenNames"
      ProcessValue <- "Tag_ScreenNumber"
      on Change: ActivateScreenByNumber("Tag_ScreenNumber", 0)
   DateTimeField "HmiScreenItemData" at 695,20 size 105x20
   DateTimeField "HmiScreenItemData_1" at 695,0 size 105x20
   GraphicView "Logo" at 0,0 size 71x40; Picture "Logo of HMI_1"

screen "Main" 800x480, template "Template_1"
   on GenerateScreen: SetTag("Tag_ScreenNumber", 1)
   TextField "Text field_1" at 319,37 size 62x32; Text 'Main'
   GraphicView "Graphic view_1" at 99,219 size 62x62; Picture "Graphic_1"
   GraphicView "Graphic view_6" at 197,168 size 105x59; Picture "Graphic_6"
      Visibility <- "Mecanisme_aplatizor"
   Rectangle "Rectangle_2" at 323,299 size 108x20
      Appearance <- "Mecanisme_forma"
   Rectangle "Rectangle_3" at 325,263 size 108x20
      Appearance <- "Mecanisme_forma"
   Rectangle "Rectangle_4" at 326,226 size 108x20
      Appearance <- "Mecanisme_forma"
   Rectangle "Rectangle_5" at 446,299 size 108x20
      Appearance <- "Mecanisme_taiere3"
   Rectangle "Rectangle_6" at 447,262 size 108x20
      Appearance <- "Mecanisme_taiere2"
   Rectangle "Rectangle_7" at 447,226 size 108x20
      Appearance <- "Mecanisme_taiere1"
   Rectangle "Rectangle_8" at 566,299 size 108x20
      Appearance <- "Mecanisme_curatare3"
   Rectangle "Rectangle_9" at 567,261 size 108x20
      Appearance <- "Mecanisme_curatare2"
   Rectangle "Rectangle_10" at 567,224 size 108x20
      Appearance <- "Mecanisme_curatare1"
   GraphicView "Graphic view_7" at 704,217 size 56x34; Picture "Graphic_9"
   Button "Button_1" at 14,145 size 42x32; TextOff 'Start'
      on Click: SetBit("Butoane_btn_start")
   SymbolicIOField "Symbolic I/O field_1" at 322,142 size 105x29; TextOff '0'; TextOn '1'; TextList "Forme"
      ProcessValue <- "Mecanisme_forma"
   TextField "Text field_2" at 336,116 size 44x20; Text 'Forma'
   TextField "Text field_3" at 101,145 size 49x20; Text 'Cuptor'
   TextField "Text field_4" at 221,128 size 64x20; Text 'Aplatizor'
   TextField "Text field_5" at 478,143 size 45x20; Text 'Taiere'
   TextField "Text field_6" at 585,144 size 63x20; Text 'Curatare'
   TextField "Text field_7" at 696,145 size 68x20; Text 'Container'
   GraphicView "Graphic view_8" at 705,256 size 56x34; Picture "Graphic_9"
   GraphicView "Graphic view_9" at 705,295 size 56x34; Picture "Graphic_9"
   Button "Button_2" at 58,368 size 47x32; TextOff 'ESD'
      on Click: SetBit("Butoane_btn_esd")
   Button "Button_3" at 59,408 size 47x32; TextOff 'Reset'
      on Click: SetBit("Butoane_reset_esd")
   Circle "Circle_1" at 65,328 size 31x31
      Appearance <- "Butoane_esd"
   IOField "I/O field_1" at 159,352 size 48x32; FormatPattern 999
      ProcessValue <- "Mecanisme_temperatura dorita la cuptor"
   IOField "I/O field_2" at 238,358 size 48x32; FormatPattern 999
      ProcessValue <- "Mecanisme_limita_c2"
   IOField "I/O field_3" at 238,397 size 48x32; FormatPattern 999
      ProcessValue <- "Mecanisme_limita_c3"
   IOField "I/O field_4" at 239,319 size 48x32; FormatPattern 999
      ProcessValue <- "Mecanisme_limita_c1"
   TextField "Text field_8" at 137,328 size 89x20; Text 'Temperatura'
   TextField "Text field_9" at 202,293 size 117x20; Text 'Limite containere'
   Circle "Circle_2" at 108,178 size 31x31
      Appearance <- "Mecanisme_cuptor"
   IOField "I/O field_5" at 711,223 size 42x23; FormatPattern 999
      ProcessValue <- "Mecanisme_container_f1"
   IOField "I/O field_6" at 713,260 size 42x23; FormatPattern 999
      ProcessValue <- "Mecanisme_container_f2"
   IOField "I/O field_7" at 712,299 size 42x23; FormatPattern 999
      ProcessValue <- "Mecanisme_container_f3"
   Button "Button_4" at 548,380 size 32x32; TextOff 'C1'
      on Click: SetBit("Butoane_golire_c1")
   Button "Button_5" at 631,379 size 32x32; TextOff 'C3'
      on Click: SetBit("Butoane_golire_c3")
   Button "Button_6" at 590,380 size 32x32; TextOff 'C2'
      on Click: SetBit("Butoane_golire_c2")
   TextField "Text field_10" at 549,355 size 116x20; Text 'Colire Containere'
   GraphicView "Graphic view_2" at 197,208 size 105x59; Picture "Graphic_6"
      Visibility <- "Mecanisme_aplatizor"
   IOField "I/O field_8" at 102,107 size 48x32; FormatPattern 999
      ProcessValue <- "Mecanisme_temperatura_cuptor"
   Button "Button_7" at 15,181 size 42x32; TextOff 'Stop'
      on Click: SetBit("Butoane_btn_start")
      on Activate: SetBit("Butoane_btn_stop")

screen "Erori interne" 800x480
   TextField "Text field_1" at 226,7 size 152x32; Text 'Erori interne'
   Button "Button_1" at 75,93 size 65x32; TextOff 'Start'
      on Click: SetBit("Avarii_avarie_start")
   Button "Button_2" at 75,137 size 65x32; TextOff 'Cuptor'
      on Click: SetBit("Avarii_avarie_cuptor")
   Button "Button_3" at 75,181 size 65x32; TextOff 'Aplatizor'
      on Click: SetBit("Avarii_avarie_aplatizor")
   Button "Button_4" at 75,225 size 65x32; TextOff 'Forme'
      on Click: SetBit("Avarii_avarie_forme")
   Button "Button_5" at 75,269 size 65x32; TextOff 'Taiere'
      on Click: SetBit("Avarii_avarie_taiere")
   Button "Button_6" at 75,313 size 65x32; TextOff 'Curatare'
      on Click: SetBit("Avarii_avarie_curatare")
   Button "Button_7" at 161,195 size 65x49; TextOff 'Reset Avarii'
      on Click: SetBit("Butoane_reset avarii")
   Circle "Circle_1" at 32,93 size 30x30
      Appearance <- "Avarii_avarie_start"
   Circle "Circle_2" at 32,314 size 30x30
      Appearance <- "Avarii_avarie_curatare"
   Circle "Circle_3" at 32,137 size 30x30
      Appearance <- "Avarii_avarie_cuptor"
   Circle "Circle_4" at 32,181 size 30x30
      Appearance <- "Avarii_avarie_aplatizor"
   Circle "Circle_5" at 32,225 size 30x30
      Appearance <- "Avarii_avarie_forme"
   Circle "Circle_6" at 32,269 size 30x30
      Appearance <- "Avarii_avarie_taiere"
*)